FUNCTION_BLOCK fbPiston EXTENDS TcoCore.TcoSequencer

METHOD PROTECTED Main : BOOL


IF Step(10,
TRUE,
'_moveHomeTask') THEN
//-------------------------------------------------------
	IF(_moveHomeTask.Invoke().Done)THEN
		StepCompleteWhen(TRUE);
	END_IF;
//-------------------------------------------------------
END_IF;

IF Step(20,
TRUE,
'_moveWorkTask') THEN
//-------------------------------------------------------
	IF(_moveWorkTask.Invoke().Done)THEN
		StepCompleteWhen(TRUE);
	END_IF;
//-------------------------------------------------------
END_IF;

IF Step(30,
TRUE,
'_moveHomeToggleTask') THEN
//-------------------------------------------------------
	IF(_moveHomeToggleTask.Toggle())THEN
		StepCompleteWhen(TRUE);
	END_IF;
//-------------------------------------------------------
END_IF;

IF Step(40,
TRUE,
'_moveHomeToggleTask') THEN
//-------------------------------------------------------
	IF(_moveHomeToggleTask.Toggle())THEN
		StepCompleteWhen(TRUE);
	END_IF;
//-------------------------------------------------------
END_IF;

IF Step(50,
TRUE,
'_moveHomeMomentaryTask') THEN
//-------------------------------------------------------
	IF(_moveHomeMomentaryTask.On())THEN
		StepCompleteWhen(TRUE);
	END_IF;
//-------------------------------------------------------
END_IF;

IF Step(60,
TRUE,
'_moveHomeMomentaryTask') THEN
//-------------------------------------------------------
	IF(_moveHomeMomentaryTask.Off())THEN
		StepCompleteWhen(TRUE);
	END_IF;
//-------------------------------------------------------
END_IF;
END_METHOD

END_FUNCTION_BLOCK

(* stored: Version 1.1.0.1, ProductVersion 3.1.4024.9
   POU fbPiston: Id {7e592838-5286-4e40-aba5-58c51ff87b0f}, SpecialFunc None
   Method Main: Id {8799706e-0a73-4966-a807-b2863f9aaaaf} *)
